METHOD PROTECTED MS_Aborting
lrHzControl := 0;
bInit := FALSE;
bRunningForward := FALSE;
bRunningReverse := FALSE;
bReset := FALSE;
bRanForward := FALSE;
bRanReverse := FALSE;
bOverLoad := FALSE;
bStop := FALSE;
bStopLog := FALSE;
bStopped := FALSE;
THIS^.tonStopDelay(IN :=FALSE);
eVfdState := VFD_UNINITIALIZED;
END_METHOD

METHOD PROTECTED MS_Idle
;
END_METHOD

METHOD  PROTECTED  MS_Initializing
// from Subclass call Super^.MS_Initializing
arrAddressWrite[iCTRL_WORD][2]	:= VFD_CTRL_RESET_FAULT;
IF eVfdStatus = VFD_STATUS_READY_TO_RUN THEN
	eVFDState := VFD_READY_INITIALIZED;
END_IF
END_METHOD

METHOD PROTECTED MS_ReadyInitialized
VAR_INPUT
END_VAR
IF NOT bInit THEN
	eVfdState := VFD_IDLE;
END_IF
END_METHOD

METHOD PROTECTED  MS_Reset
VAR_INPUT
END_VAR
arrAddressWrite[iCTRL_WORD][2]	:= VFD_CTRL_RESET_FAULT;
IF THIS^.evfdStatus <>  VFD_STATUS_NOT_RESPOND AND
	THIS^.evfdStatus <>  VFD_STATUS_FAULT THEN
	evfdState := VFD_RESET_DONE;
END_IF
END_METHOD

METHOD PROTECTED MS_ResetDone
VAR_INPUT
END_VAR
IF NOT bReset THEN
	evfdState := VFD_IDLE;
END_IF
END_METHOD

METHOD PROTECTED  MS_RunForward
VAR_INPUT
END_VAR
(*arrAddressWrite[iCtrlFrequencyWord][2] :=  LREAL_TO_WORD( 
											FC_ScaleValue(		rangeRawMin := 0,
																rangeRawMax := 50,
																RangeScaleMin := WORD_TO_LREAL( wHzWordValueMin),
																RangeScaleMax := WORD_TO_LREAL( wHzWordValueMax),
																ValueRaw := lrHzControl) 
														);*)
arrAddressWrite[iCTRL_WORD][2]	:= VFD_CTRL_RUN_FORWARD;
IF eVfdStatus = VFD_STATUS_RUNNING_FORWARD 
(*AND F_InRange( bound1 := lrHzControl + 1,
				bound2 := lrHzControl -1,
				value := lrHzActual)*)
THEN
	eVFDState := VFD_RUN_FORWARD_DONE;
END_IF
END_METHOD

METHOD PROTECTED MS_RunForwardDone
IF NOT bRunningForward THEN
	eVfdState := VFD_IDLE;
END_IF
END_METHOD

METHOD PROTECTED  MS_RunReverse
VAR_INPUT
END_VAR
(*arrAddressWrite[iCtrlFrequencyWord][2] :=  LREAL_TO_WORD( 
											FC_ScaleValue(		rangeRawMin := 0,
																rangeRawMax := 50,
																RangeScaleMin := WORD_TO_LREAL( wHzWordValueMin),
																RangeScaleMax := WORD_TO_LREAL( wHzWordValueMax),
																ValueRaw := lrHzControl) 
														);*)
arrAddressWrite[iCTRL_WORD][2]	:= VFD_CTRL_RUN_REVERSE;
IF eVfdStatus = VFD_STATUS_RUNNING_REVERSE 
(*AND F_InRange( bound1 := lrHzControl + 1,
				bound2 := lrHzControl -1,
				value := lrHzActual)*)
THEN
	eVFDState := VFD_RUN_REVERSE_DONE;
END_IF
END_METHOD

METHOD PROTECTED MS_RunReverseDone
VAR_INPUT
END_VAR
IF NOT bRunningReverse THEN
	eVfdState := VFD_IDLE;
END_IF
END_METHOD

METHOD protected  MS_Stop 
VAR_INPUT
END_VAR
arrAddressWrite[iCTRL_WORD][2]	:= VFD_CTRL_STOP_SPEED_DOWN;
(*tonStopDelay( in := eVfdStatus = VFD_STATUS_STOP,
				PT := tStopDelay);*)
IF eVfdStatus = VFD_STATUS_STOP THEN
 eVfdState := VFD_STOP_DONE;	
END_IF
(*IF tonStopDelay.Q THEN
	tonStopDelay(IN := FALSE);
	
END_IF*)
END_METHOD

METHOD protected Ms_StopDone
VAR_INPUT
END_VAR
IF NOT bStop THEN
	eVfdState := VFD_IDLE;
END_IF
END_METHOD

METHOD PROTECTED MS_Uninitialized
END_METHOD

{attribute 'monitoring' := 'variable'}
PROPERTY Overload : reference TO BOOL
GET
Overload REF= bOverLoad;
END_GET
END_PROPERTY

{attribute 'monitoring' := 'variable'}
PROPERTY PowerKw : REFERENCE TO LREAL
GET
PowerKw ref= lrPowerKw;
END_GET
END_PROPERTY

PROPERTY Speed : Reference to lreal
GET
Speed REF= lrSpeed;
END_GET
END_PROPERTY

{attribute 'monitoring' := 'variable'}
PROPERTY State : reference to E_Vfd_State
GET
State REF= eVfdState;
END_GET
END_PROPERTY

METHOD PROTECTED StateMachine
CASE eVfdState OF
	VFD_UNINITIALIZED :
		MS_Uninitialized();
		
	VFD_INITIALIZING	:
		MS_Initializing();
		
	VFD_READY_INITIALIZED :
		MS_ReadyInitialized();
		
	VFD_IDLE:
		MS_Idle();
	
	VFD_RUN_FORWARD	:
		MS_RunForward();
		
	VFD_RUN_FORWARD_DONE:
		MS_RunForwardDone();
	
	VFD_RUN_REVERSE	:
		MS_RunReverse();
	
	VFD_RUN_REVERSE_DONE:
		MS_RunReverseDone();
	
	VFD_STOP		:
		MS_Stop();
		
	VFD_STOP_DONE	:
		Ms_StopDone();
		
	VFD_RESET	:
		MS_Reset();
		
	VFD_RESET_DONE	:
		MS_ResetDone();
		
	VFD_ABORTING :
		MS_Aborting();
	
	
END_CASE
END_METHOD

{attribute 'monitoring' := 'variable'}
PROPERTY Status : reference to E_VFD_Status
GET
Status REF= eVfdStatus;
END_GET
END_PROPERTY

PROPERTY timeStopDelay : time
GET
timeStopDelay := THIS^.tStopDelay;
END_GET
SET
tStopDelay := timeStopDelay;
END_SET
END_PROPERTY

PROPERTY Torque : reference to lreal
GET
Torque ref= Torque;
END_GET
END_PROPERTY

PROPERTY TotalKwh : reference to lreal
GET
TotalKwh REF= TotalKwh;
END_GET
END_PROPERTY

// not all vfd modbus available this function 
PROPERTY Warning : reference to bool
GET
Warning  ref= bWarning;
END_GET
END_PROPERTY

END_FUNCTION_BLOCK

// ---- POUs/VFD/FB_VFD_ABB_ACS480.TcPOU
FUNCTION_BLOCK FB_VFD_ABB_ACS480 EXTENDS FB_UniversalVFDModbus

VAR
	VFD_CTRL_RUN_EMERGENCY_STOP : WORD;
	TempData0: U_Word2Int;
END_VAR

SUPER^();

METHOD Convert : BOOL
VAR_INPUT
	iRegionNo	:	INT;
	pReadData	:	POINTER TO word;
END_VAR
CASE	iRegionNo OF

	0: // status
		IF pReadData[0].15 = TRUE THEN
			eVfdStatus := VFD_STATUS_FAULT;
			
		ELSIF (eVfdState = VFD_INITIALIZING
			OR eVfdState = VFD_READY_INITIALIZED)
			AND pReadData[0].0 = TRUE
			AND pReadData[0].1 = TRUE	
			AND pReadData[0].2 = TRUE
			THEN
			eVfdStatus :=  VFD_STATUS_READY_TO_RUN;
				
		ELSIF pReadData[0].3 = FALSE THEN
			eVfdStatus :=  VFD_STATUS_STOP;
			
		ELSIF pReadData[0].3 = TRUE	//run
			AND pReadData[0].10 = FALSE	// Drive reference is in the forward direction	
			AND pReadData[0].11 = FALSE//Drive is running in the forward direction
			THEN		
			eVfdStatus := VFD_STATUS_RUNNING_FORWARD;
		
		ELSIF pReadData[0].3 = TRUE	//run
			AND pReadData[0].10 = TRUE	// Drive reference is in the forward direction	
			AND pReadData[0].11 = TRUE//Drive is running in the forward direction
			THEN		
			eVfdStatus := VFD_STATUS_RUNNING_REVERSE;
		
		END_IF
	1: 
		TempData0.iWord := pReadData[0];
		lrHzActual		:= ABS(INT_TO_LREAL( TempData0.iInt)*0.0025);//50/20000;	
		lrCurrent		:= WORD_TO_LREAL( pReadData[1])*0.01;	//46.05 = 100
		lrDcVoltage		:= WORD_TO_LREAL( pReadData[5])*0.1;	
	
	2: 
		lrVacOutToMotor	:= WORD_TO_LREAL( pReadData[0]);	//4099	/1
		lrPowerKw		:= WORD_TO_LREAL( pReadData[1])*0.01;		//46.04
	
	3:
		lrTotalKwh :=  WORD_TO_LREAL( pReadData[0])*0.1;
		
	4: 
		lrSpeed :=  WORD_TO_LREAL( pReadData[0]);
	
	


END_CASE
END_METHOD

METHOD  FirstCycle 
VAR_INPUT
	sName : STRING;
	iUnitID : BYTE ; // modbus address of the device : 1- 255
END_VAR
SUPER^.FirstCycle( sName := sName, iUnitID := iUnitID);
(*Assign Ctrol Word : user Manual M-driver*)
VFD_CTRL_RESET_FAULT := 2#0001_0001;
VFD_CTRL_RUN_FORWARD := 2#0000_0010;
VFD_CTRL_RUN_REVERSE := 2#0000_0110;
VFD_CTRL_STOP_FREE 	 := 2#0010_0000_0001;
VFD_CTRL_STOP_SPEED_DOWN := 2#1000_0001;
VFD_CTRL_RUN_EMERGENCY_STOP := 2#0001_0000_0001;

// actual state	
	arrAddressRead[0][0] := 3;
	arrAddressRead[0][1] := 1;
	arrAddressRead[0][2] := E_ModbusFunction.ReadHoldingRegisters;

//mode0 address = 40000 + function*100 + sub function -1
	// actual hz  
	arrAddressRead[1][0] := 105; // 01.06
	arrAddressRead[1][1] := 6;
	arrAddressRead[1][2] := E_ModbusFunction.ReadHoldingRegisters;
	
	arrAddressRead[2][0] := 112; // 01.13
	arrAddressRead[2][1] := 2;
	arrAddressRead[2][2] := E_ModbusFunction.ReadHoldingRegisters;
	
	arrAddressRead[3][0] := 119; // 01.20
	arrAddressRead[3][1] := 1;
	arrAddressRead[3][2] := E_ModbusFunction.ReadHoldingRegisters;
	
	arrAddressRead[4][0] := 101; // 01.20
	arrAddressRead[4][1] := 1;
	arrAddressRead[4][2] := E_ModbusFunction.ReadHoldingRegisters;
iNumAddRegionRead	:= 5;

/////write control WORD VFD, // use ctrol word and frequency in 1 modbus write
arrAddressWrite[iCTRL_WORD][0]	:= 0;
arrAddressWrite[iCTRL_WORD][1]	:= 2;
arrAddressWrite[iCTRL_WORD][2]	:= VFD_CTRL_STOP_FREE;
arrAddressWrite[iCTRL_WORD][10]	:= E_ModbusFunction.WriteMultipleRegisters;

// Frequency
//arrAddressWrite[iCTRL_FREQUENCY_WORD][0]	:= 1;
//arrAddressWrite[iCTRL_FREQUENCY_WORD][1]	:= 1;
							(*MUST BE CARE FULL WHEN USE FLOATING POINT CONVERT*)
arrAddressWrite[iCTRL_FREQUENCY_WORD][3]	:= LREAL_TO_WORD( F_ScaleValue(	rangeRawMin := 0,
																				rangeRawMax := 50,
																				RangeScaleMin :=0,
																				RangeScaleMax := 20000,
																				ValueRaw := 0)
										  );
										  
iNumAddRegionWrite := 1;// use ctrol word and frequency in 1 modbus write
END_METHOD

METHOD PROTECTED  MS_Aborting
arrAddressWrite[iCTRL_WORD][2]	:= VFD_CTRL_STOP_FREE;
SUPER^.MS_Aborting();
END_METHOD

METHOD  PROTECTED  MS_Initializing
SUPER^.MS_Initializing();
END_METHOD

METHOD PROTECTED  MS_RunForward
VAR_INPUT
END_VAR
// use ctrol word and frequency in 1 modbus write WRITE MULTIES REGIS
arrAddressWrite[iCTRL_WORD][3] :=  LREAL_TO_WORD( 
															F_ScaleValue(	rangeRawMin := 0,
																			rangeRawMax := 50,
																			RangeScaleMin := 0,
																			RangeScaleMax := 20000,
																			ValueRaw := lrHzControl) 
																				);
SUPER^.MS_RunForward();
END_METHOD

METHOD PROTECTED  MS_RunReverse
VAR_INPUT
END_VAR
// use ctrol word and frequency in 1 modbus write WRITE MULTIES REGIS
arrAddressWrite[iCTRL_WORD][3] :=  LREAL_TO_WORD( 
															F_ScaleValue(	rangeRawMin := 0,
																			rangeRawMax := 50,
																			RangeScaleMin := 0,
																			RangeScaleMax := 20000,
																			ValueRaw := lrHzControl) 
																				);
SUPER^.MS_RunReverse();
END_METHOD

END_FUNCTION_BLOCK

// ---- POUs/VFD/FB_VFD_Mdriver.TcPOU
FUNCTION_BLOCK FB_VFD_Mdriver EXTENDS FB_UniversalVFDModbus

VAR
	eFaultInfor	: E_VfdMdriverFaultInfor;
END_VAR

//bError := eVfdStatus
SUPER^();

METHOD Convert : BOOL
VAR_INPUT
	iRegionNo	:	INT;
	pReadData	:	POINTER TO word;
END_VAR
CASE	iRegionNo OF
	0: 
	
		lrHzActual		:= WORD_TO_LREAL( pReadData[0])*0.01;	//4097	/unit /100
		lrDcVoltage		:= WORD_TO_LREAL( pReadData[1])*0.1;	//4098 	/10
		lrVacOutToMotor	:= WORD_TO_LREAL( pReadData[2]);	//4099	/1
		lrCurrent		:= WORD_TO_LREAL(  pReadData[3])*0.01;		//4100	/100
		//4 reserve
		lrPowerKw		:= WORD_TO_LREAL(  pReadData[5])*0.001;		//4102	/1000> kW
	
	1: // status
		CASE pReadData[0] OF
			0: eVfdStatus := VFD_STATUS_STOP;
			
			1: 
				eVfdStatus := VFD_STATUS_RUNNING_FORWARD;
			2:
				eVfdStatus := VFD_STATUS_RUNNING_REVERSE;
			3: 
				eVfdStatus := VFD_STATUS_STOP;
		END_CASE
		// important
		IF eVfdState = VFD_INITIALIZING THEN
			IF eFaultInfor = E_VfdMdriverFaultInfor.Nofault
			AND eVfdStatus = VFD_STATUS_STOP THEN
				eVfdStatus := VFD_STATUS_READY_TO_RUN;
			ELSIF eFaultInfor <> E_VfdMdriverFaultInfor.Nofault THEN
				eVfdStatus := VFD_STATUS_FAULT;
			END_IF
		END_IF
		IF eFaultInfor <> E_VfdMdriverFaultInfor.Nofault THEN
			eVfdStatus := VFD_STATUS_FAULT;
		END_IF
		IF iModbusErrorID = MODBUSERROR_C_NO_RESPONSE THEN
			eVfdStatus := VFD_STATUS_NOT_RESPOND;
		END_IF
		// important
	
	2: 
	
		iErrorID := WORD_TO_UDINT( pReadData[0]);
		eFaultInfor :=  WORD_TO_UINT( pReadData[0]);
END_CASE
END_METHOD

METHOD  FirstCycle 
VAR_INPUT
	sName : STRING;
	iUnitID : BYTE ; // modbus address of the device : 1- 255
END_VAR
SUPER^.FirstCycle( sName := sName, iUnitID := iUnitID);
(*Assign Ctrol Word : user Manual M-driver*)
VFD_CTRL_RESET_FAULT := 7;
VFD_CTRL_RUN_FORWARD := 1;
VFD_CTRL_RUN_REVERSE := 2;
VFD_CTRL_STOP_FREE 		:= 5;
VFD_CTRL_STOP_SPEED_DOWN	:= 6;
///  actual hz, current, voltage
arrAddressRead[0][0] := 4097;
arrAddressRead[0][1]	:= 6;
arrAddressRead[0][2]	:= E_ModbusFunction.ReadHoldingRegisters;

// actual state	
arrAddressRead[1][0] := 16#3000;
arrAddressRead[1][1]	:= 1;
arrAddressRead[1][2]	:= E_ModbusFunction.ReadHoldingRegisters;

// fault infor
arrAddressRead[2][0] := 16#8000;
arrAddressRead[2][1]	:= 1;
arrAddressRead[2][2]	:= E_ModbusFunction.ReadHoldingRegisters;

iNumAddRegionRead	:= 3;

/////write control WORD VFD
arrAddressWrite[iCTRL_WORD][0]	:= 16#2000;
arrAddressWrite[iCTRL_WORD][1]	:= 1;
arrAddressWrite[iCTRL_WORD][2]	:= VFD_CTRL_STOP_FREE;
arrAddressWrite[iCTRL_WORD][10]	:= E_ModbusFunction.WriteSingleRegister;
// Frequency
arrAddressWrite[iCTRL_FREQUENCY_WORD][0]	:= 4096;
arrAddressWrite[iCTRL_FREQUENCY_WORD][1]	:= 1;
							(*MUST BE CARE FULL WHEN USE FLOATING POINT CONVERT*)
arrAddressWrite[iCTRL_FREQUENCY_WORD][2]	:= LREAL_TO_WORD( F_ScaleValue(	rangeRawMin := 0,
															rangeRawMax := 50,
															RangeScaleMin :=0,
															RangeScaleMax := 10000,
															ValueRaw := 0)
										  );
arrAddressWrite[iCTRL_FREQUENCY_WORD][10]	:= E_ModbusFunction.WriteSingleRegister;
										  
iNumAddRegionWrite := 2;
END_METHOD

METHOD PROTECTED  MS_Aborting
arrAddressWrite[iCTRL_WORD][2]	:= VFD_CTRL_STOP_FREE;
SUPER^.MS_Aborting();
END_METHOD

METHOD PROTECTED  MS_RunForward
VAR_INPUT
END_VAR
arrAddressWrite[iCTRL_FREQUENCY_WORD][2] :=  LREAL_TO_WORD( 
															F_ScaleValue(	rangeRawMin := 0,
																			rangeRawMax := 50,
																			RangeScaleMin := 0,
																			RangeScaleMax := 10000,
																			ValueRaw := lrHzControl) 
																				);
SUPER^.MS_RunForward();
END_METHOD

METHOD PROTECTED  MS_RunReverse
VAR_INPUT
END_VAR
arrAddressWrite[iCTRL_FREQUENCY_WORD][2] :=  LREAL_TO_WORD( 
															F_ScaleValue(	rangeRawMin := 0,
																			rangeRawMax := 50,
																			RangeScaleMin := 0,
																			RangeScaleMax := 10000,
																			ValueRaw := lrHzControl) 
																				);
SUPER^.MS_RunReverse();
END_METHOD

END_FUNCTION_BLOCK

// ---- POUs/VFD/FB_VFD_V20_Siemens.TcPOU
FUNCTION_BLOCK FB_VFD_V20_Siemens EXTENDS FB_UniversalVFDModbus
VAR			
	// status word
	Inverter_Ready		: BOOL;
	InverterReadyToRun	: BOOL;
	InverterRunning		: BOOL;
	InverterFaultActive : BOOL;
	OFF2_active			: BOOL;
	OFF3_active			: BOOL;
	ON_inhibit_active 	 : BOOL;
	Inverter_warning_active : BOOL;
	Deviation_setpoint_OR_ActiveValue : BOOL;
	PZD_control 		: BOOL;
	Motor_current_Or_torque_limit  : BOOL;
	Brake_open	 : BOOL;
	Motor_overload : BOOL;
	Motor_RunRight	: BOOL;
	Inverter_overload :BOOL; 
	//mode
	///  actual  Speed ( rpm) (unit A : Scale factor 1), Current ( A , 100, , Torque (Nm, 100)
	//, Actual Power (kw, 100), Total Kwh( 1), Dc bus Voltage(1), REFERENCE( hz, 100), RATED PWR( 100),OUTPUT VOLTS(1)
END_VAR

SUPER^();

METHOD Convert : BOOL
VAR_INPUT
	iRegionNo	:	INT;
	pReadData	:	POINTER TO word;
END_VAR
CASE iRegionNo OF
	0:
		// Status word
		Inverter_Ready		:=  pReadData[0].0;
		InverterReadyToRun	:=  pReadData[0].1;
		InverterRunning		:=  pReadData[0].2;
		InverterFaultActive :=  pReadData[0].3;
		OFF2_active			:= NOT pReadData[0].4;
		OFF3_active			:= NOT  pReadData[0].5;
		ON_inhibit_active 	 := pReadData[0].6;
		Inverter_warning_active := pReadData[0].7;
		Deviation_setpoint_OR_ActiveValue := NOT pReadData[0].8;
		PZD_control 		:= pReadData[0].9;
		Motor_current_Or_torque_limit  := NOT pReadData[0].11;
		Brake_open	 := pReadData[0].12;
		Motor_overload := NOT pReadData[0].13;
		Motor_RunRight	:= pReadData[0].14;
		Inverter_overload :=  NOT pReadData[0].15;
		
		IF eVfdState = VFD_INITIALIZING AND Inverter_Ready THEN
			eVfdStatus := VFD_STATUS_READY_TO_RUN;
		ELSIF InverterFaultActive THEN
			eVfdStatus := VFD_STATUS_FAULT;
//		ELSIF InverterFaultActive THEN
//			eVfdStatus := VFD_STATUS_WARNING;
		ELSIF InverterRunning THEN
			IF Motor_RunRight THEN
				eVfdStatus := VFD_STATUS_RUNNING_FORWARD;
			ELSE
				eVfdStatus := VFD_STATUS_RUNNING_REVERSE;
			END_IF
		ELSIF NOT InverterRunning THEN
			eVfdStatus := VFD_STATUS_STOP;
		END_IF

		// Speed word
		lrHzactual := WORD_TO_LREAL( pReadData[1])*50/16383;
		
	1:
		///  actual  Speed ( rpm) (unit A : Scale factor 1), Current ( A , 100, , Torque (Nm, 100)
	//, Actual Power (kw, 100), Total Kwh( 1), Dc bus Voltage(1), REFERENCE( hz, 100), RATED PWR( 100),OUTPUT VOLTS(1)
		lrSpeed := pReadData[0];
		lrCurrent := WORD_TO_LREAL(pReadData[1])/100;
		lrTorque := WORD_TO_LREAL(pReadData[2])/100;
		lrPowerKw := WORD_TO_LREAL(pReadData[3])/100;
		lrTotalKwh := WORD_TO_LREAL(pReadData[4]);
		lrDcVoltage := WORD_TO_LREAL(pReadData[5]);
		lrRatedPower := WORD_TO_LREAL(pReadData[7])/100;
		lrVACOutToMotor := WORD_TO_LREAL(pReadData[8]);
END_CASE
END_METHOD

METHOD  FirstCycle 
VAR_INPUT
	sName : STRING;
	iUnitID : BYTE ; // modbus address of the device : 1- 255
END_VAR
THIS^.sName := sName;
THIS^.iUnitID := iUnitID;
VFD_CTRL_STOP_FREE		:= 2#010001111010; // casue fault , reset error to run again	
VFD_CTRL_RUN_FORWARD	:= 2#010001111111;	
VFD_CTRL_RUN_REVERSE	 := 2#110001111111;	
VFD_CTRL_STOP_SPEED_DOWN := 2#010001111110;
VFD_CTRL_RESET_FAULT	 := 2#010011111110;
(*HSW (speed setpoint), HIW (actual speed), STW (control word), ZSW (status word) refer to
control data. For more information, see parameters r2018 and P2019 in Chapter "Parameter
list (Page 147)*)

//ZSW  (status WORD), HIW (actual speed)
	arrAddressRead[0][0] := 109;
	arrAddressRead[0][1] := 2;
	arrAddressRead[0][2] := E_ModbusFunction.ReadHoldingRegisters;
///  actual  Speed ( rpm) (unit A : Scale factor 1), Current ( A , 100, , Torque (Nm, 100)
	//, Actual Power (kw, 100), Total Kwh( 1), Dc bus Voltage(1), REFERENCE( hz, 100), RATED PWR( 100),OUTPUT VOLTS(1)
	arrAddressRead[1][0] := 24;
	arrAddressRead[1][1] := 10;
	arrAddressRead[1][2] := E_ModbusFunction.ReadHoldingRegisters;
	
iNumAddRegionRead	:= 2;
/////write control  VFD
// Control word																	
arrAddressWrite[iCTRL_WORD][0]	:= 99;
arrAddressWrite[iCTRL_WORD][1]  := 1;
arrAddressWrite[iCTRL_WORD][2]	:= 1150; //VFD_CTRL_STOP_SPEED_DOWN
arrAddressWrite[iCTRL_WORD][10]	:= E_ModbusFunction.WriteSingleRegister;	
// Frequency
arrAddressWrite[iCTRL_FREQUENCY_WORD][0]	:= 100;
arrAddressWrite[iCTRL_FREQUENCY_WORD][1] 	:= 1;
arrAddressWrite[iCTRL_FREQUENCY_WORD][2]	:= LREAL_TO_WORD( F_ScaleValue(	rangeRawMin := 0,
																				rangeRawMax := 50,
																				RangeScaleMin :=0,
																				RangeScaleMax := 16384,
																				ValueRaw := lrHzControl)
															 );
arrAddressWrite[iCTRL_FREQUENCY_WORD][10]	:= E_ModbusFunction.WriteSingleRegister;												
iNumAddRegionWrite := 2;
END_METHOD

METHOD PROTECTED MS_Aborting
arrAddressWrite[iCTRL_WORD][2] := VFD_CTRL_STOP_FREE;
SUPER^.MS_Aborting();
END_METHOD

METHOD PROTECTED  MS_RunForward
VAR_INPUT
END_VAR
arrAddressWrite[iCTRL_FREQUENCY_WORD][2] :=  LREAL_TO_WORD( F_ScaleValue(	rangeRawMin := 0,
																			rangeRawMax := 50,
																			RangeScaleMin :=0,
																			RangeScaleMax := 16384,
																			ValueRaw := lrHzControl) );
SUPER^.MS_RunForward();
END_METHOD

METHOD PROTECTED  MS_RunReverse
VAR_INPUT
END_VAR
arrAddressWrite[iCTRL_FREQUENCY_WORD][2] :=  LREAL_TO_WORD( F_ScaleValue(	rangeRawMin := 0,
																			rangeRawMax := 50,
																			RangeScaleMin :=0,
																			RangeScaleMax := 16384,
																			ValueRaw := lrHzControl) );
super^.MS_RunReverse();
END_METHOD

END_FUNCTION_BLOCK

// ---- TEST/PGR_Test.TcPOU
PROGRAM PGR_Test
VAR
	fbUniversalVfdModbusTest : FB_UniversalVFDModbus_Test;
	fbvfd : FB_VFD_ABB_ACS480;
END_VAR

TcUnit.RUN();

END_PROGRAM
